// TIA Portal project "Selector" (V16)

(* hardware
DEVICE "S7-1200 station_1"  S7-1200 Station
   slot 0: "Rack_0"  S7-1200 Rack  Rack  V1.0
   slot 1: "PLC_1"  CPU 1212C AC/DC/Rly  6ES7 212-1BE40-0XB0  V4.0
*)

// ===== PLC "PLC_1"  CPU 1212C AC/DC/Rly =====

VAR_GLOBAL   // PLC tag table "Default tag table"
   "k1" AT %Q0.0 : Bool;
   "X1" AT %M1.0 : Bool;
   "X2" AT %M1.1 : Bool;
   "X3" AT %M1.2 : Bool;
   "K2" AT %Q0.1 : Bool;
   "K3" AT %Q0.2 : Bool;
   "selector2" AT %I0.5 : Bool;
   "selector1" AT %I0.4 : Bool;
   "Tag_1" AT %M2.3 : Bool;
   "Tag_4" AT %M5.3 : Bool;
   "Tag_5" AT %M5.4 : Bool;
   "Tag_6" AT %M5.5 : Bool;
   "Tag_7" AT %M5.6 : Bool;
   "Tag_8" AT %M5.1 : Bool;
   "Tag_9" AT %M5.2 : Bool;
   "Tag_10" AT %I0.1 : Bool;
   "Tag_11" AT %I0.3 : Bool;
   "Tag_12" AT %M6.0 : Bool;
END_VAR

// folder: System blocks/Program resources

DATA_BLOCK "T1"   // DB1
{ S7_Optimized_Access := 'TRUE' }
AUTHOR : Simatic
FAMILY : IEC
NAME : IEC_TMR
VERSION : 1.0
// stored: InstanceOfName IEC_TIMER
"IEC_TIMER"
BEGIN
END_DATA_BLOCK

DATA_BLOCK "T2"   // DB2
{ S7_Optimized_Access := 'TRUE' }
AUTHOR : Simatic
FAMILY : IEC
NAME : IEC_TMR
VERSION : 1.0
// stored: InstanceOfName IEC_TIMER
"IEC_TIMER"
BEGIN
END_DATA_BLOCK

// folder: (top level)

ORGANIZATION_BLOCK "Main"   // OB1, LAD, ProgramCycle
TITLE = "Main Program Sweep (Cycle)"
{ S7_Optimized_Access := 'TRUE' }
VERSION : 0.1
   VAR_INPUT
      Initial_Call : Bool;   // Initial call of this OB
      Remanence : Bool;   // =True, if remanent data are available
   END_VAR
BEGIN

REGION Network 1
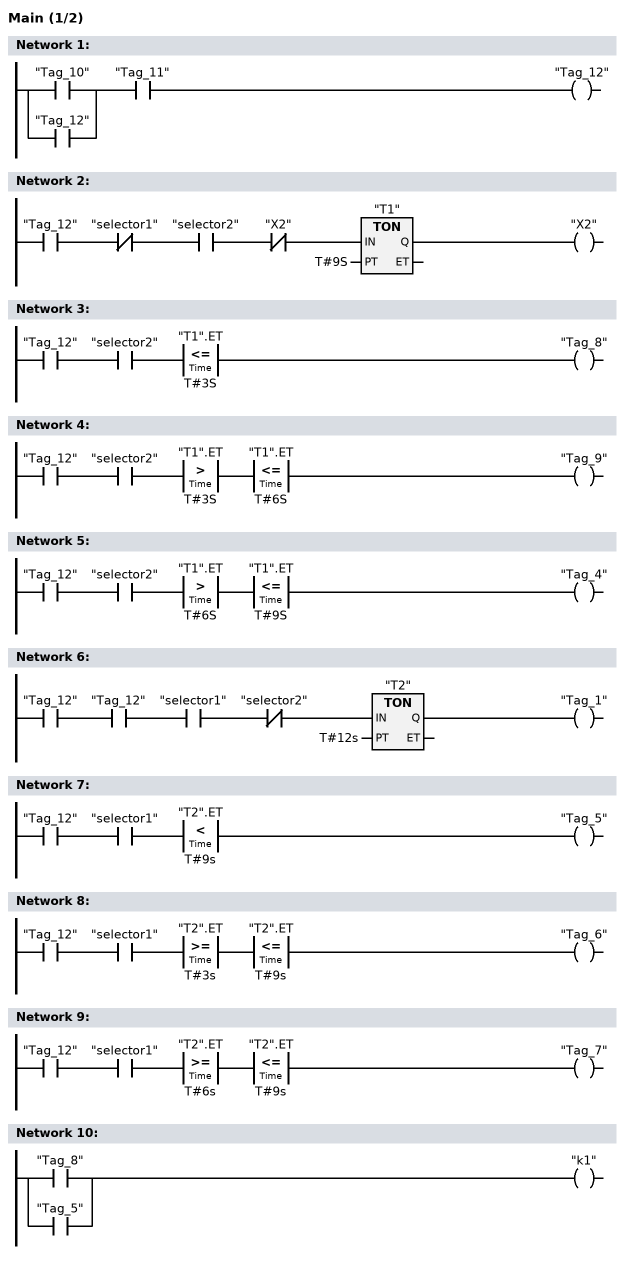
   RUNG wire#powerrail
      Contact( "Tag_10" )
      wire#w1
      Contact( "Tag_11" )
      Coil( "Tag_12" )
   END_RUNG
   RUNG wire#powerrail
      Contact( "Tag_12" )
   END_RUNG wire#w1
   // the same network as SCL:
   "Tag_12" := ("Tag_10" OR "Tag_12") AND "Tag_11";
END_REGION

REGION Network 2
   "T1".TON(IN := "Tag_12" AND NOT "selector1" AND "selector2" AND NOT "X2", PT := T#9S);
   "X2" := "T1".Q;
END_REGION

REGION Network 3
   RUNG wire#powerrail
      Contact( "Tag_12" )
      Contact( "selector2" )
      { S7_Templates := "SrcType := Time" } LE_Contact(in1 := "T1".ET, in2 := T#3S)
      Coil( "Tag_8" )
   END_RUNG
   // the same network as SCL:
   "Tag_8" := "Tag_12" AND "selector2" AND ("T1".ET <= T#3S);
END_REGION

REGION Network 4
   RUNG wire#powerrail
      Contact( "Tag_12" )
      Contact( "selector2" )
      { S7_Templates := "SrcType := Time" } GT_Contact(in1 := "T1".ET, in2 := T#3S)
      { S7_Templates := "SrcType := Time" } LE_Contact(in1 := "T1".ET, in2 := T#6S)
      Coil( "Tag_9" )
   END_RUNG
   // the same network as SCL:
   "Tag_9" := "Tag_12" AND "selector2" AND ("T1".ET > T#3S) AND ("T1".ET <= T#6S);
END_REGION

REGION Network 5
   RUNG wire#powerrail
      Contact( "Tag_12" )
      Contact( "selector2" )
      { S7_Templates := "SrcType := Time" } GT_Contact(in1 := "T1".ET, in2 := T#6S)
      { S7_Templates := "SrcType := Time" } LE_Contact(in1 := "T1".ET, in2 := T#9S)
      Coil( "Tag_4" )
   END_RUNG
   // the same network as SCL:
   "Tag_4" := "Tag_12" AND "selector2" AND ("T1".ET > T#6S) AND ("T1".ET <= T#9S);
END_REGION

REGION Network 6
   "T2".TON(IN := "Tag_12" AND "Tag_12" AND "selector1" AND NOT "selector2", PT := T#12s);
   "Tag_1" := "T2".Q;
END_REGION

REGION Network 7
   RUNG wire#powerrail
      Contact( "Tag_12" )
      Contact( "selector1" )
      { S7_Templates := "SrcType := Time" } LT_Contact(in1 := "T2".ET, in2 := T#9s)
      Coil( "Tag_5" )
   END_RUNG
   // the same network as SCL:
   "Tag_5" := "Tag_12" AND "selector1" AND ("T2".ET < T#9s);
END_REGION

REGION Network 8
   RUNG wire#powerrail
      Contact( "Tag_12" )
      Contact( "selector1" )
      { S7_Templates := "SrcType := Time" } GE_Contact(in1 := "T2".ET, in2 := T#3s)
      { S7_Templates := "SrcType := Time" } LE_Contact(in1 := "T2".ET, in2 := T#9s)
      Coil( "Tag_6" )
   END_RUNG
   // the same network as SCL:
   "Tag_6" := "Tag_12" AND "selector1" AND ("T2".ET >= T#3s) AND ("T2".ET <= T#9s);
END_REGION

REGION Network 9
   RUNG wire#powerrail
      Contact( "Tag_12" )
      Contact( "selector1" )
      { S7_Templates := "SrcType := Time" } GE_Contact(in1 := "T2".ET, in2 := T#6s)
      { S7_Templates := "SrcType := Time" } LE_Contact(in1 := "T2".ET, in2 := T#9s)
      Coil( "Tag_7" )
   END_RUNG
   // the same network as SCL:
   "Tag_7" := "Tag_12" AND "selector1" AND ("T2".ET >= T#6s) AND ("T2".ET <= T#9s);
END_REGION

REGION Network 10
   RUNG wire#powerrail
      Contact( "Tag_8" )
      wire#w1
      Coil( "k1" )
   END_RUNG
   RUNG wire#powerrail
      Contact( "Tag_5" )
   END_RUNG wire#w1
   // the same network as SCL:
   "k1" := "Tag_8" OR "Tag_5";
END_REGION

REGION Network 11
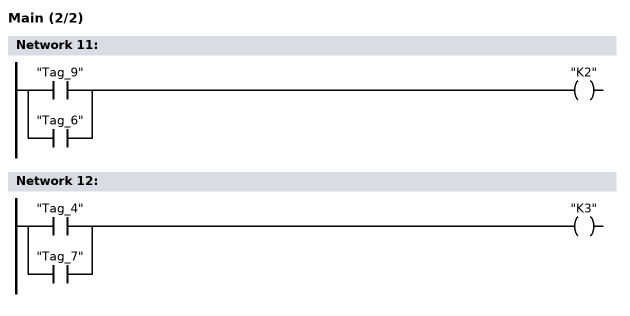
   RUNG wire#powerrail
      Contact( "Tag_9" )
      wire#w1
      Coil( "K2" )
   END_RUNG
   RUNG wire#powerrail
      Contact( "Tag_6" )
   END_RUNG wire#w1
   // the same network as SCL:
   "K2" := "Tag_9" OR "Tag_6";
END_REGION

REGION Network 12
   RUNG wire#powerrail
      Contact( "Tag_4" )
      wire#w1
      Coil( "K3" )
   END_RUNG
   RUNG wire#powerrail
      Contact( "Tag_7" )
   END_RUNG wire#w1
   // the same network as SCL:
   "K3" := "Tag_4" OR "Tag_7";
END_REGION
END_ORGANIZATION_BLOCK